{attribute 'GeneratedUsingTerminal: EK1814-0000-0016'}
{attribute addProperty BoxType "EK1814-0000-0016"}
{attribute addProperty Id "InputAT %I*BOOL1"}
{attribute addProperty CRC "2198356929"}
{attribute addProperty Size "1"}
TYPE Channel_830843C1 EXTENDS DigitalInputBase_50022E7B :
STRUCT
	{attribute addProperty Name "Input"}
	Input AT %I* : BOOL;
END_STRUCT
END_TYPE

(* stored: Version 1.2.0.0, ProductVersion 3.1.4024.9
   DUT Channel_830843C1: Id {ccd79baa-2d7c-4264-833b-ad297f76232c} *)
